// TIA Portal V18 export
// export: Created 2026-01-09T11:23:29.8932705Z, ExportSetting WithDefaults, DisplayName Totally Integrated Automation Portal, DisplayVersion V18 Update 5, DisplayName TIA Portal Openness, DisplayVersion V18 Update 5, DisplayName TIA Portal Teamcenter Gateway, DisplayVersion V18, DisplayName TIA Portal Version Control Interface, DisplayVersion V18, DisplayName SINAMICS Startdrive Advanced, DisplayVersion V18 SP2 Update 1, DisplayName SINAMICS Startdrive G110M, G120, G120C, G120D, G120P, G115D, DisplayVersion V18 SP2 Update 1, DisplayName SINAMICS Startdrive G130, G150, S120, S150, SINAMICS MV, S210, G220, S200, DisplayVersion V18 SP2 Update 1, DisplayName STEP 7 Professional, DisplayVersion V18 Update 5, DisplayName STEP 7 Safety, DisplayVersion V18, DisplayName WinCC Professional, DisplayVersion V18 Update 5
Screen "218 Scanner_803A1"  1280x800, Number=218, Template=02ManualUnit1
  ScreenLayer "Layer_0"
    FaceplateInstance "RCS_fpKeyenceSR1000_TP1200_1" at 30,148 size 1102x383  FaceplateTypeName=KeyenceSR1000@$@03_FacePlate@$@RCS_fpKeyenceSR1000_TP1200 V 0.0.8
      InterfacePropertyText "文本"  Text="803A1_RingScan"
      Property := KeyenceSR1000Ctrl_803A1DB_sHMI
    Button "btnMenu8_7" at 383,725 size 128x75  Mode=Text, TextOff="A-读码器 803A1 / A-CodeReader 803A1", TextOn="A-读码器 803A1 / A-CodeReader 803A1"
      RangeAppearanceAnimation "RangeAppearanceAnimation"
        tag 
        0..0: back #636571, fore #000000
        1..1: back #0000ff, fore #000000
      on Click: ActivateScreen(Screen name := , Object number := 0)
    Button "btnMenu6" at 640,725 size 128x75  Mode=Text
    Button "btnMenu7" at 896,725 size 128x75  Mode=Text
    Button "btnMenu6_1" at 768,725 size 128x75  Mode=Text
    Button "btnMenu7_1" at 1024,725 size 128x75  Mode=Text, TextOff="上一页 / PreviousPage", TextOn="上一页 / PreviousPage"
      on Click: ActivateScreen(Screen name := 210_Cylinder_A1, Object number := 0)
    Button "按钮_1" at 256,725 size 128x75  Mode=Text, TextOff="A-伺服 383A1 / A-Servo 383A1", TextOn="A-伺服 383A1 / A-Servo 383A1"
      on Click: ActivateScreen(Screen name := 217-Servo_383A1, Object number := 0)
    Button "按钮_2" at 511,725 size 128x75  Mode=Text, PictureOff=向右箭头_0, TextOff="A-读码器 802A1 / A-CodeReader 802A1", TextOn="A-读码器 802A1 / A-CodeReader 802A1"
      RangeAppearanceAnimation "RangeAppearanceAnimation"
        tag ST_CommandTestLamp
        1..1: back #00ff00, fore #000000
      on Click: ActivateScreen(Screen name := 219 X80Scanner_802A1, Object number := 0)
    Button "btnMenu8_4" at 127,725 size 128x75  Mode=Text, TextOff="A-气缸2 / A-Cylinder2", TextOn="A-气缸2 / A-Cylinder2"
      on Click: ActivateScreen(Screen name := 216_Cylinder_A2, Object number := 0)
